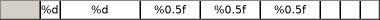
VISUALIZATION _VISU_RepeatHistoryEntry  // 380x20
VAR_IN_OUT
	mInst : ST_RepeatHistory;
END_VAR
    RoundedRectangle (0,0 40x20), colour toggle: mInst.bSelected
    Rectangle (40,0 20x20), "%d", text variable: mInst.nIndex
    Rectangle (60,0 80x20), "%d", tooltip "X0 [SubPx]", text variable: mInst.nX0
    Rectangle (140,0 60x20), "%0.5f", tooltip "Length Effective", text variable: mInst.fLenEffective
    Rectangle (200,0 60x20), "%0.5f", tooltip "Length Configured", text variable: mInst.fLen
    Rectangle (260,0 60x20), "%0.5f", tooltip "Length diff", text variable: mInst.fLenDiff
    RoundedRectangle (320,0 20x20), tooltip "Length not in range", colour toggle: mInst.bLenNotInRange
    RoundedRectangle (340,0 20x20), tooltip "invalid & ignored marks", colour toggle: mInst.bInvalidIngoredMarks
    RoundedRectangle (360,0 20x20), tooltip "missing marks", colour toggle: mInst.bMissingMarks
END_VISUALIZATION

(* stored: Version 1.1.0.1, ProductVersion 3.1.4024.11
   Visu _VISU_RepeatHistoryEntry: Id {b7e555da-1d75-41a7-aa0f-f0ee0f89641a} *)
